TYPE aut_location:
    (l1_aut_location, l2_aut_location);
END_TYPE

(* stored: ProductVersion 3.1.0.18, Version 1.1.0.1 *)
